// An enum that can be used to represent getters and setters.
TYPE FsT_Accessor : FsE_Accessor; END_TYPE

(* stored: Version 1.1.0.1, ProductVersion 3.1.4024.4
   DUT FsT_Accessor: Id {fcfc1be2-dec2-4f16-b7b5-e433e5688cd7} *)
